FUNCTION F_PistonDisplacementToBoomAngle : LREAL
VAR_INPUT
	xCyl : LREAL;
END_VAR
VAR
	AB : LREAL;
	AC : LREAL;
	BC : LREAL;
	alpha1 : LREAL;
	alpha2 : LREAL;
	theta1 : LREAL;
	AB2 : LREAL;
	AC2 : LREAL;
	BC2 : LREAL;
END_VAR

AB := SQRT(ABS(Parameters.stParam.stCraneKinematics.ABx)*ABS(Parameters.stParam.stCraneKinematics.ABx) + ABS(Parameters.stParam.stCraneKinematics.ABy)*ABS(Parameters.stParam.stCraneKinematics.ABy));
AC := SQRT(ABS(Parameters.stParam.stCraneKinematics.ACx)*ABS(Parameters.stParam.stCraneKinematics.ACx) + ABS(Parameters.stParam.stCraneKinematics.ACy)*ABS(Parameters.stParam.stCraneKinematics.ACy));

BC := 0.77222 + xCyl;

alpha1 := ATAN(ABS(Parameters.stParam.stCraneKinematics.ACy)/ ABS(Parameters.stParam.stCraneKinematics.ACx));
alpha2 := ATAN(ABS(Parameters.stParam.stCraneKinematics.ABy)/ ABS(Parameters.stParam.stCraneKinematics.ABx));

AB2 := ABS(AB)*ABS(AB);
AC2 := ABS(AC)*ABS(AC);
BC2 := ABS(BC)*ABS(BC);

theta1 := ACOS( (AB2 + AC2 - BC2) / (2 * ABS(AB) * ABS(AC)) ) - alpha2 + alpha1;

F_PistonDisplacementToBoomAngle := theta1;

END_FUNCTION

(* stored: Version 1.1.0.1, ProductVersion 3.1.4024.10
   POU F_PistonDisplacementToBoomAngle: Id {a235119c-45d2-4f49-b730-4da55738c20e}, SpecialFunc None *)
